SUBAPPLICATION Ventilsteuerung_Uebung_012c (* String Input und Speichern (WIP) *)
  (* Standard: 61499-2 *)
  (* Version 1.0, 2023-10-23, franz *)
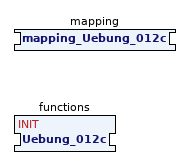
  SUBAPPS
    mapping : mapping_Uebung_012c;
    functions : Uebung_012c;
  END_SUBAPPS
END_SUBAPPLICATION
